// Mitsubishi GX Works2 project: Class7_Ex01(컨베이어&실린더)   PLC: Q03UD

PROGRAM MAIN
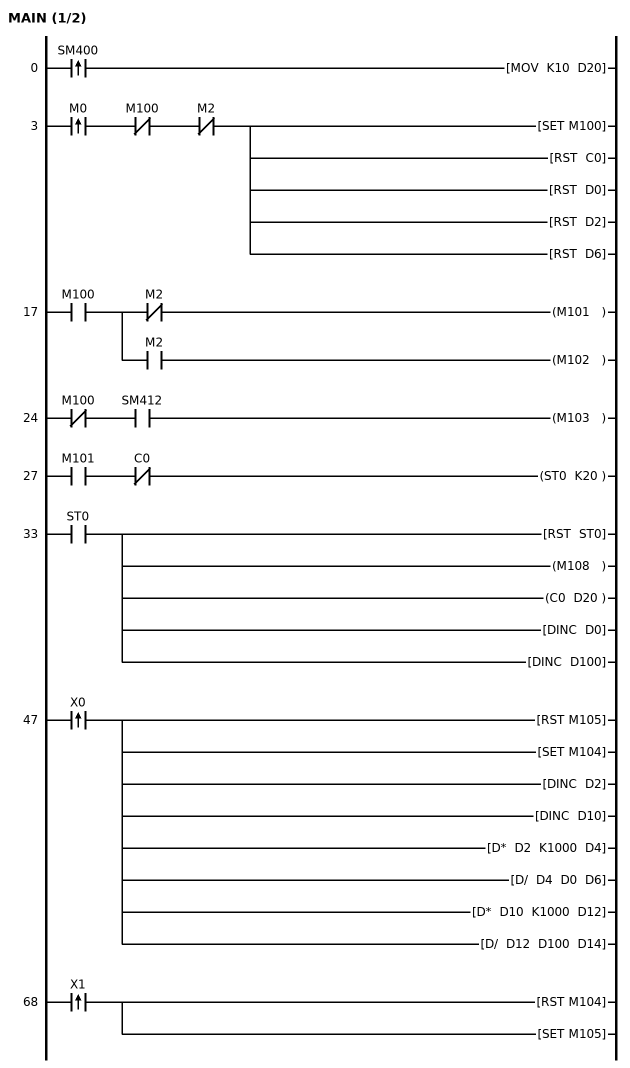
0     LDP     SM400
      MOV     K10 D20
3     LDP     M0
      ANI     M100
      ANI     M2
      SET     M100
      RST     C0
      RST     D0
      RST     D2
      RST     D6
17    LD      M100
      MPS
      ANI     M2
      OUT     M101
      MPP
      AND     M2
      OUT     M102
24    LDI     M100
      AND     SM412
      OUT     M103
27    LD      M101
      ANI     C0
      OUT     ST0 K20
33    LD      ST0
      RST     ST0
      OUT     M108
      OUT     C0 D20
      DINC    D0
      DINC    D100
47    LDP     X0
      RST     M105
      SET     M104
      DINC    D2
      DINC    D10
      D*      D2 K1000 D4
      D/      D4 D0 D6
      D*      D10 K1000 D12
      D/      D12 D100 D14
68    LDP     X1
      RST     M104
      SET     M105
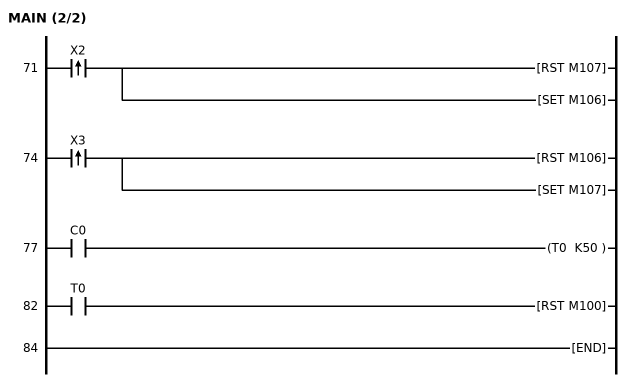
71    LDP     X2
      RST     M107
      SET     M106
74    LDP     X3
      RST     M106
      SET     M107
77    LD      C0
      OUT     T0 K50
82    LD      T0
      RST     M100
84    END
END_PROGRAM
